// TIA Portal V16 export
// export: Created 2023-03-29T11:03:29.1138509Z, ExportSetting WithDefaults, DisplayName Totally Integrated Automation Portal, DisplayVersion V16 Update 6, DisplayName TIA Portal Version Control Interface, DisplayVersion V16 Update 2, DisplayName TIA Portal Openness, DisplayVersion V16 Update 6, DisplayName STEP 7 Professional, DisplayVersion V16 Update 6, DisplayName STEP 7 Safety, DisplayVersion V16, DisplayName WinCC Advanced, DisplayVersion V16 Update 6
FUNCTION "Sterowniki napędów" : Void   // FC7, LAD
TITLE = Sterowniki
{ S7_Optimized_Access := 'TRUE' }
AUTHOR : rtecmer
VERSION : 0.1
// Sterownik napędów zasuw Z1-Z9
// stored: AutoNumber true, IsIECCheckEnabled false, SetENOAutomatically false, UDAEnableTagReadback false
BEGIN

REGION Network 2: Sterowanie Zasuwą Z10 - Położenie
   // Funkcja zawiera kontrolę czasu jazdy na pozycję ustawiony czas 120sek
   // po upływie czasu nastapi alarm i przełączenie w trym manual
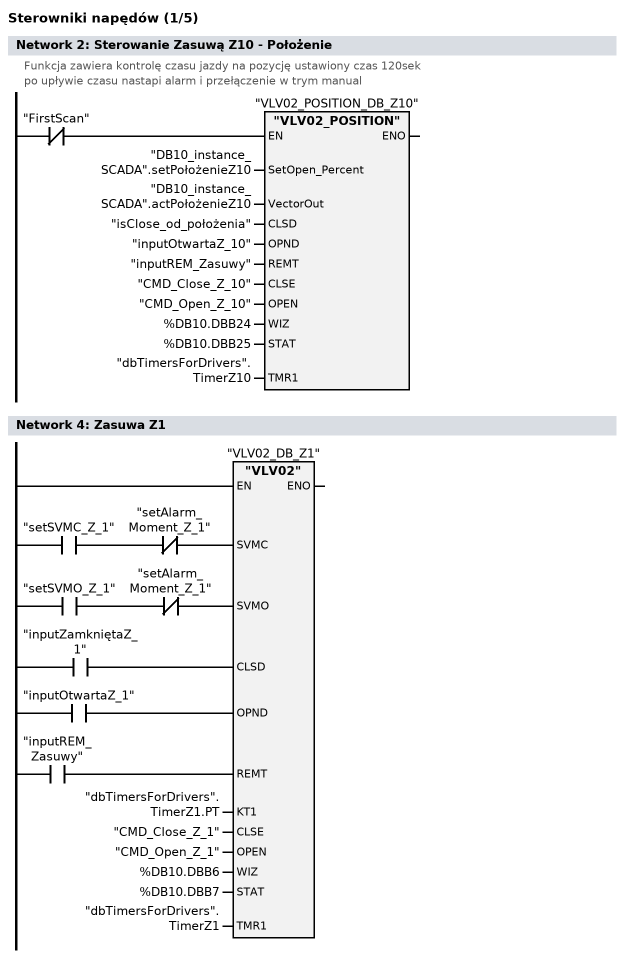
   RUNG wire#powerrail
      I_Contact( "FirstScan" )
      "VLV02_POSITION_DB_Z10"(SetOpen_Percent := "DB10_instance_SCADA".setPołożenieZ10, VectorOut := "DB10_instance_SCADA".actPołożenieZ10, CLSD := "isClose_od_położenia", OPND := "inputOtwartaZ_10", REMT := "inputREM_Zasuwy", CLSE := "CMD_Close_Z_10", OPEN := "CMD_Open_Z_10", WIZ := %DB10.DBB24, STAT := %DB10.DBB25, TMR1 := "dbTimersForDrivers".TimerZ10)
   END_RUNG
   // the same network as SCL:
   IF NOT "FirstScan" THEN
       "VLV02_POSITION_DB_Z10"(SetOpen_Percent := "DB10_instance_SCADA".setPołożenieZ10,   // "VLV02_POSITION"
                               VectorOut := "DB10_instance_SCADA".actPołożenieZ10,
                               CLSD := "isClose_od_położenia",
                               OPND := "inputOtwartaZ_10",
                               REMT := "inputREM_Zasuwy",
                               CLSE := "CMD_Close_Z_10",
                               OPEN := "CMD_Open_Z_10",
                               WIZ := %DB10.DBB24,
                               STAT := %DB10.DBB25,
                               TMR1 := "dbTimersForDrivers".TimerZ10);
   END_IF;
END_REGION

REGION Network 4: Zasuwa Z1
   RUNG wire#powerrail
      "VLV02_DB_Z1"(SVMC := wire#w1, SVMO := wire#w2, CLSD := wire#w3, OPND := wire#w4, REMT := wire#w5, KT1 := "dbTimersForDrivers".TimerZ1.PT, CLSE := "CMD_Close_Z_1", OPEN := "CMD_Open_Z_1", WIZ := %DB10.DBB6, STAT := %DB10.DBB7, TMR1 := "dbTimersForDrivers".TimerZ1)
   END_RUNG
   RUNG wire#powerrail
      Contact( "setSVMC_Z_1" )
      I_Contact( "setAlarm_Moment_Z_1" )
   END_RUNG wire#w1
   RUNG wire#powerrail
      Contact( "setSVMO_Z_1" )
      I_Contact( "setAlarm_Moment_Z_1" )
   END_RUNG wire#w2
   RUNG wire#powerrail
      Contact( "inputZamkniętaZ_1" )
   END_RUNG wire#w3
   RUNG wire#powerrail
      Contact( "inputOtwartaZ_1" )
   END_RUNG wire#w4
   RUNG wire#powerrail
      Contact( "inputREM_Zasuwy" )
   END_RUNG wire#w5
   // the same network as SCL:
   "VLV02_DB_Z1"(SVMC := "setSVMC_Z_1" AND NOT "setAlarm_Moment_Z_1",   // "VLV02"
                 SVMO := "setSVMO_Z_1" AND NOT "setAlarm_Moment_Z_1",
                 CLSD := "inputZamkniętaZ_1",
                 OPND := "inputOtwartaZ_1",
                 REMT := "inputREM_Zasuwy",
                 KT1 := "dbTimersForDrivers".TimerZ1.PT,
                 CLSE := "CMD_Close_Z_1",
                 OPEN := "CMD_Open_Z_1",
                 WIZ := %DB10.DBB6,
                 STAT := %DB10.DBB7,
                 TMR1 := "dbTimersForDrivers".TimerZ1);
END_REGION

REGION Network 5: Zasuwa Z2
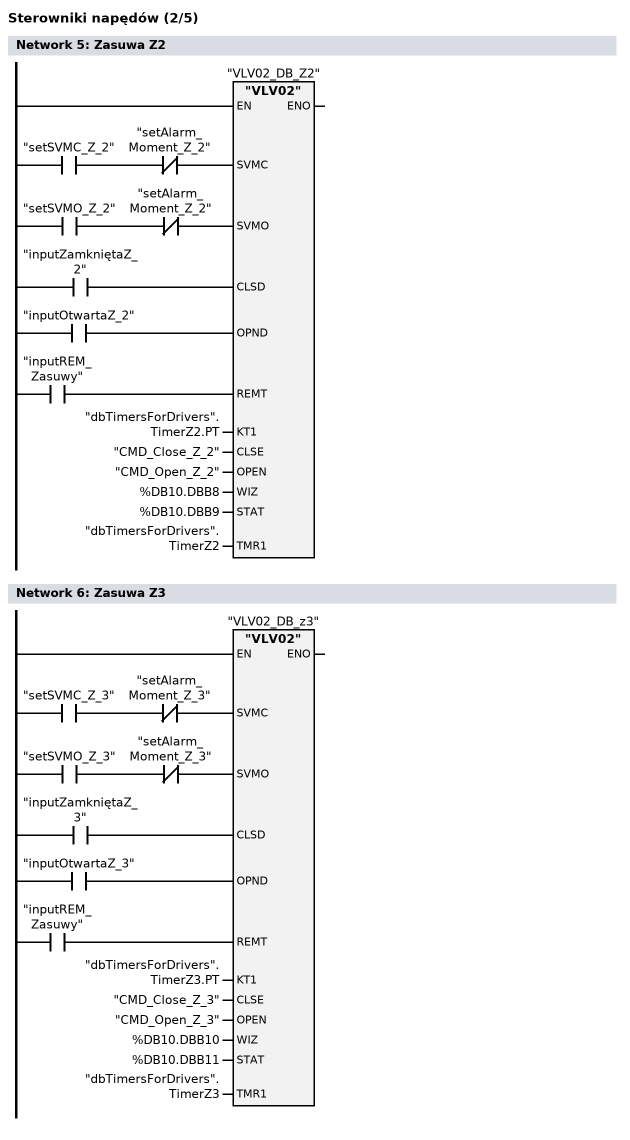
   RUNG wire#powerrail
      "VLV02_DB_Z2"(SVMC := wire#w1, SVMO := wire#w2, CLSD := wire#w3, OPND := wire#w4, REMT := wire#w5, KT1 := "dbTimersForDrivers".TimerZ2.PT, CLSE := "CMD_Close_Z_2", OPEN := "CMD_Open_Z_2", WIZ := %DB10.DBB8, STAT := %DB10.DBB9, TMR1 := "dbTimersForDrivers".TimerZ2)
   END_RUNG
   RUNG wire#powerrail
      Contact( "setSVMC_Z_2" )
      I_Contact( "setAlarm_Moment_Z_2" )
   END_RUNG wire#w1
   RUNG wire#powerrail
      Contact( "setSVMO_Z_2" )
      I_Contact( "setAlarm_Moment_Z_2" )
   END_RUNG wire#w2
   RUNG wire#powerrail
      Contact( "inputZamkniętaZ_2" )
   END_RUNG wire#w3
   RUNG wire#powerrail
      Contact( "inputOtwartaZ_2" )
   END_RUNG wire#w4
   RUNG wire#powerrail
      Contact( "inputREM_Zasuwy" )
   END_RUNG wire#w5
   // the same network as SCL:
   "VLV02_DB_Z2"(SVMC := "setSVMC_Z_2" AND NOT "setAlarm_Moment_Z_2",   // "VLV02"
                 SVMO := "setSVMO_Z_2" AND NOT "setAlarm_Moment_Z_2",
                 CLSD := "inputZamkniętaZ_2",
                 OPND := "inputOtwartaZ_2",
                 REMT := "inputREM_Zasuwy",
                 KT1 := "dbTimersForDrivers".TimerZ2.PT,
                 CLSE := "CMD_Close_Z_2",
                 OPEN := "CMD_Open_Z_2",
                 WIZ := %DB10.DBB8,
                 STAT := %DB10.DBB9,
                 TMR1 := "dbTimersForDrivers".TimerZ2);
END_REGION

REGION Network 6: Zasuwa Z3
   RUNG wire#powerrail
      "VLV02_DB_z3"(SVMC := wire#w1, SVMO := wire#w2, CLSD := wire#w3, OPND := wire#w4, REMT := wire#w5, KT1 := "dbTimersForDrivers".TimerZ3.PT, CLSE := "CMD_Close_Z_3", OPEN := "CMD_Open_Z_3", WIZ := %DB10.DBB10, STAT := %DB10.DBB11, TMR1 := "dbTimersForDrivers".TimerZ3)
   END_RUNG
   RUNG wire#powerrail
      Contact( "setSVMC_Z_3" )
      I_Contact( "setAlarm_Moment_Z_3" )
   END_RUNG wire#w1
   RUNG wire#powerrail
      Contact( "setSVMO_Z_3" )
      I_Contact( "setAlarm_Moment_Z_3" )
   END_RUNG wire#w2
   RUNG wire#powerrail
      Contact( "inputZamkniętaZ_3" )
   END_RUNG wire#w3
   RUNG wire#powerrail
      Contact( "inputOtwartaZ_3" )
   END_RUNG wire#w4
   RUNG wire#powerrail
      Contact( "inputREM_Zasuwy" )
   END_RUNG wire#w5
   // the same network as SCL:
   "VLV02_DB_z3"(SVMC := "setSVMC_Z_3" AND NOT "setAlarm_Moment_Z_3",   // "VLV02"
                 SVMO := "setSVMO_Z_3" AND NOT "setAlarm_Moment_Z_3",
                 CLSD := "inputZamkniętaZ_3",
                 OPND := "inputOtwartaZ_3",
                 REMT := "inputREM_Zasuwy",
                 KT1 := "dbTimersForDrivers".TimerZ3.PT,
                 CLSE := "CMD_Close_Z_3",
                 OPEN := "CMD_Open_Z_3",
                 WIZ := %DB10.DBB10,
                 STAT := %DB10.DBB11,
                 TMR1 := "dbTimersForDrivers".TimerZ3);
END_REGION

REGION Network 7: Zasuwa Z4
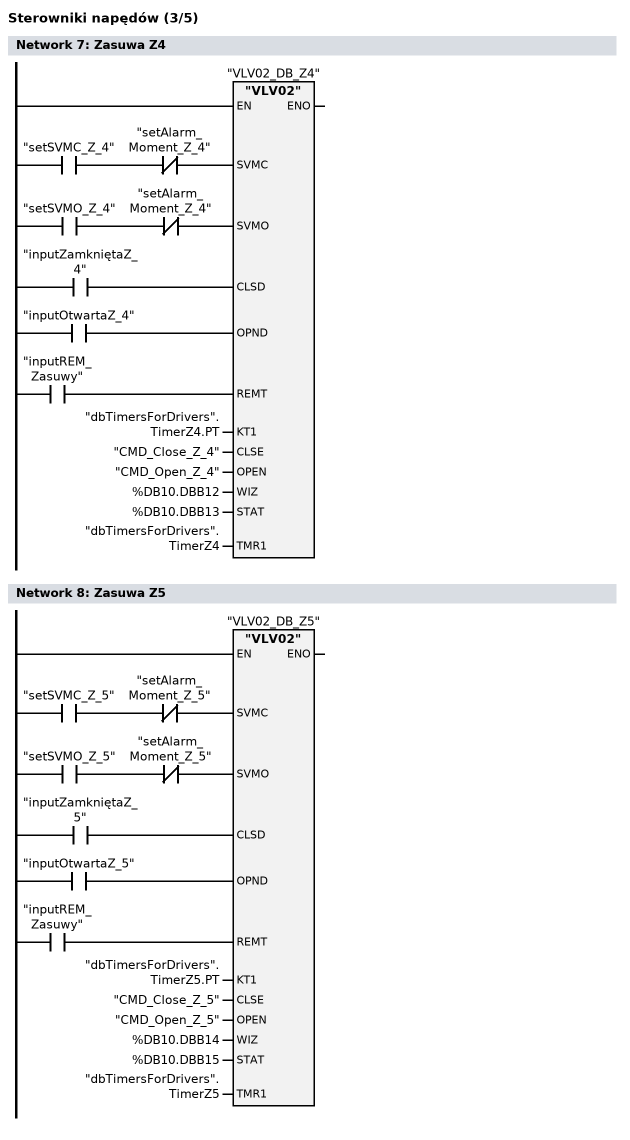
   RUNG wire#powerrail
      "VLV02_DB_Z4"(SVMC := wire#w1, SVMO := wire#w2, CLSD := wire#w3, OPND := wire#w4, REMT := wire#w5, KT1 := "dbTimersForDrivers".TimerZ4.PT, CLSE := "CMD_Close_Z_4", OPEN := "CMD_Open_Z_4", WIZ := %DB10.DBB12, STAT := %DB10.DBB13, TMR1 := "dbTimersForDrivers".TimerZ4)
   END_RUNG
   RUNG wire#powerrail
      Contact( "setSVMC_Z_4" )
      I_Contact( "setAlarm_Moment_Z_4" )
   END_RUNG wire#w1
   RUNG wire#powerrail
      Contact( "setSVMO_Z_4" )
      I_Contact( "setAlarm_Moment_Z_4" )
   END_RUNG wire#w2
   RUNG wire#powerrail
      Contact( "inputZamkniętaZ_4" )
   END_RUNG wire#w3
   RUNG wire#powerrail
      Contact( "inputOtwartaZ_4" )
   END_RUNG wire#w4
   RUNG wire#powerrail
      Contact( "inputREM_Zasuwy" )
   END_RUNG wire#w5
   // the same network as SCL:
   "VLV02_DB_Z4"(SVMC := "setSVMC_Z_4" AND NOT "setAlarm_Moment_Z_4",   // "VLV02"
                 SVMO := "setSVMO_Z_4" AND NOT "setAlarm_Moment_Z_4",
                 CLSD := "inputZamkniętaZ_4",
                 OPND := "inputOtwartaZ_4",
                 REMT := "inputREM_Zasuwy",
                 KT1 := "dbTimersForDrivers".TimerZ4.PT,
                 CLSE := "CMD_Close_Z_4",
                 OPEN := "CMD_Open_Z_4",
                 WIZ := %DB10.DBB12,
                 STAT := %DB10.DBB13,
                 TMR1 := "dbTimersForDrivers".TimerZ4);
END_REGION

REGION Network 8: Zasuwa Z5
   RUNG wire#powerrail
      "VLV02_DB_Z5"(SVMC := wire#w1, SVMO := wire#w2, CLSD := wire#w3, OPND := wire#w4, REMT := wire#w5, KT1 := "dbTimersForDrivers".TimerZ5.PT, CLSE := "CMD_Close_Z_5", OPEN := "CMD_Open_Z_5", WIZ := %DB10.DBB14, STAT := %DB10.DBB15, TMR1 := "dbTimersForDrivers".TimerZ5)
   END_RUNG
   RUNG wire#powerrail
      Contact( "setSVMC_Z_5" )
      I_Contact( "setAlarm_Moment_Z_5" )
   END_RUNG wire#w1
   RUNG wire#powerrail
      Contact( "setSVMO_Z_5" )
      I_Contact( "setAlarm_Moment_Z_5" )
   END_RUNG wire#w2
   RUNG wire#powerrail
      Contact( "inputZamkniętaZ_5" )
   END_RUNG wire#w3
   RUNG wire#powerrail
      Contact( "inputOtwartaZ_5" )
   END_RUNG wire#w4
   RUNG wire#powerrail
      Contact( "inputREM_Zasuwy" )
   END_RUNG wire#w5
   // the same network as SCL:
   "VLV02_DB_Z5"(SVMC := "setSVMC_Z_5" AND NOT "setAlarm_Moment_Z_5",   // "VLV02"
                 SVMO := "setSVMO_Z_5" AND NOT "setAlarm_Moment_Z_5",
                 CLSD := "inputZamkniętaZ_5",
                 OPND := "inputOtwartaZ_5",
                 REMT := "inputREM_Zasuwy",
                 KT1 := "dbTimersForDrivers".TimerZ5.PT,
                 CLSE := "CMD_Close_Z_5",
                 OPEN := "CMD_Open_Z_5",
                 WIZ := %DB10.DBB14,
                 STAT := %DB10.DBB15,
                 TMR1 := "dbTimersForDrivers".TimerZ5);
END_REGION

REGION Network 9: Zasuwa Z6
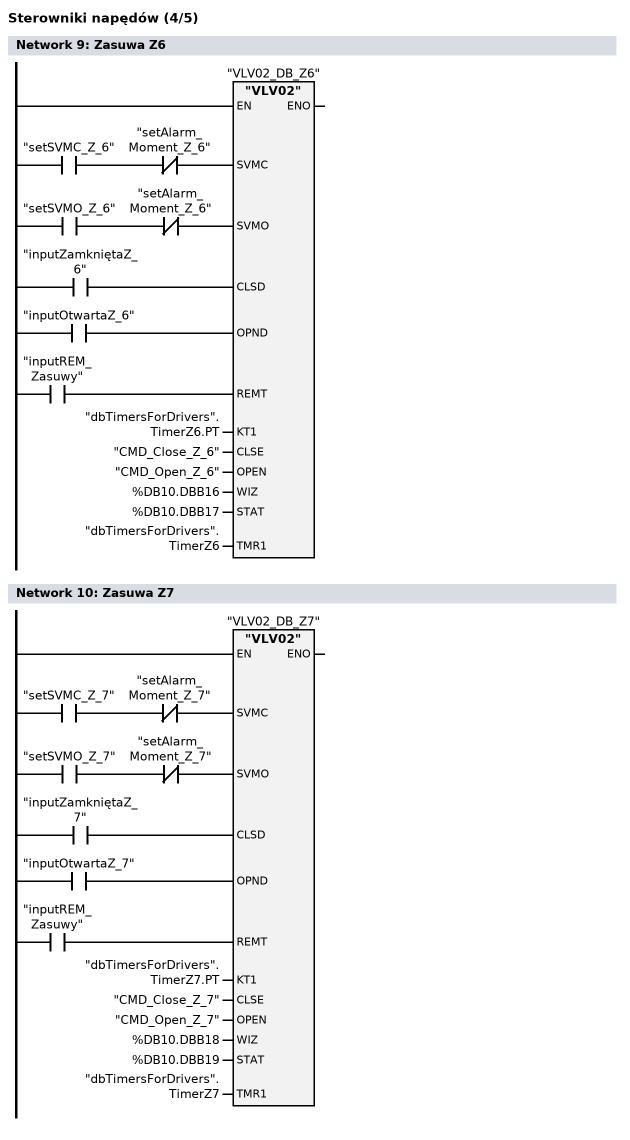
   RUNG wire#powerrail
      "VLV02_DB_Z6"(SVMC := wire#w1, SVMO := wire#w2, CLSD := wire#w3, OPND := wire#w4, REMT := wire#w5, KT1 := "dbTimersForDrivers".TimerZ6.PT, CLSE := "CMD_Close_Z_6", OPEN := "CMD_Open_Z_6", WIZ := %DB10.DBB16, STAT := %DB10.DBB17, TMR1 := "dbTimersForDrivers".TimerZ6)
   END_RUNG
   RUNG wire#powerrail
      Contact( "setSVMC_Z_6" )
      I_Contact( "setAlarm_Moment_Z_6" )
   END_RUNG wire#w1
   RUNG wire#powerrail
      Contact( "setSVMO_Z_6" )
      I_Contact( "setAlarm_Moment_Z_6" )
   END_RUNG wire#w2
   RUNG wire#powerrail
      Contact( "inputZamkniętaZ_6" )
   END_RUNG wire#w3
   RUNG wire#powerrail
      Contact( "inputOtwartaZ_6" )
   END_RUNG wire#w4
   RUNG wire#powerrail
      Contact( "inputREM_Zasuwy" )
   END_RUNG wire#w5
   // the same network as SCL:
   "VLV02_DB_Z6"(SVMC := "setSVMC_Z_6" AND NOT "setAlarm_Moment_Z_6",   // "VLV02"
                 SVMO := "setSVMO_Z_6" AND NOT "setAlarm_Moment_Z_6",
                 CLSD := "inputZamkniętaZ_6",
                 OPND := "inputOtwartaZ_6",
                 REMT := "inputREM_Zasuwy",
                 KT1 := "dbTimersForDrivers".TimerZ6.PT,
                 CLSE := "CMD_Close_Z_6",
                 OPEN := "CMD_Open_Z_6",
                 WIZ := %DB10.DBB16,
                 STAT := %DB10.DBB17,
                 TMR1 := "dbTimersForDrivers".TimerZ6);
END_REGION

REGION Network 10: Zasuwa Z7
   RUNG wire#powerrail
      "VLV02_DB_Z7"(SVMC := wire#w1, SVMO := wire#w2, CLSD := wire#w3, OPND := wire#w4, REMT := wire#w5, KT1 := "dbTimersForDrivers".TimerZ7.PT, CLSE := "CMD_Close_Z_7", OPEN := "CMD_Open_Z_7", WIZ := %DB10.DBB18, STAT := %DB10.DBB19, TMR1 := "dbTimersForDrivers".TimerZ7)
   END_RUNG
   RUNG wire#powerrail
      Contact( "setSVMC_Z_7" )
      I_Contact( "setAlarm_Moment_Z_7" )
   END_RUNG wire#w1
   RUNG wire#powerrail
      Contact( "setSVMO_Z_7" )
      I_Contact( "setAlarm_Moment_Z_7" )
   END_RUNG wire#w2
   RUNG wire#powerrail
      Contact( "inputZamkniętaZ_7" )
   END_RUNG wire#w3
   RUNG wire#powerrail
      Contact( "inputOtwartaZ_7" )
   END_RUNG wire#w4
   RUNG wire#powerrail
      Contact( "inputREM_Zasuwy" )
   END_RUNG wire#w5
   // the same network as SCL:
   "VLV02_DB_Z7"(SVMC := "setSVMC_Z_7" AND NOT "setAlarm_Moment_Z_7",   // "VLV02"
                 SVMO := "setSVMO_Z_7" AND NOT "setAlarm_Moment_Z_7",
                 CLSD := "inputZamkniętaZ_7",
                 OPND := "inputOtwartaZ_7",
                 REMT := "inputREM_Zasuwy",
                 KT1 := "dbTimersForDrivers".TimerZ7.PT,
                 CLSE := "CMD_Close_Z_7",
                 OPEN := "CMD_Open_Z_7",
                 WIZ := %DB10.DBB18,
                 STAT := %DB10.DBB19,
                 TMR1 := "dbTimersForDrivers".TimerZ7);
END_REGION

REGION Network 11: Zasuwa Z8
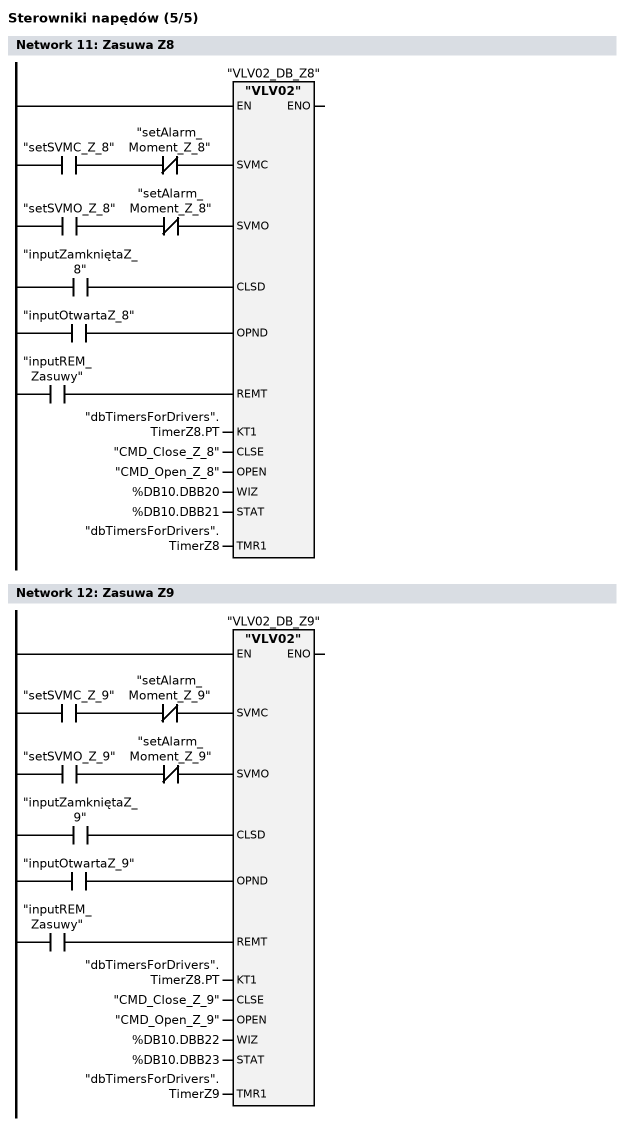
   RUNG wire#powerrail
      "VLV02_DB_Z8"(SVMC := wire#w1, SVMO := wire#w2, CLSD := wire#w3, OPND := wire#w4, REMT := wire#w5, KT1 := "dbTimersForDrivers".TimerZ8.PT, CLSE := "CMD_Close_Z_8", OPEN := "CMD_Open_Z_8", WIZ := %DB10.DBB20, STAT := %DB10.DBB21, TMR1 := "dbTimersForDrivers".TimerZ8)
   END_RUNG
   RUNG wire#powerrail
      Contact( "setSVMC_Z_8" )
      I_Contact( "setAlarm_Moment_Z_8" )
   END_RUNG wire#w1
   RUNG wire#powerrail
      Contact( "setSVMO_Z_8" )
      I_Contact( "setAlarm_Moment_Z_8" )
   END_RUNG wire#w2
   RUNG wire#powerrail
      Contact( "inputZamkniętaZ_8" )
   END_RUNG wire#w3
   RUNG wire#powerrail
      Contact( "inputOtwartaZ_8" )
   END_RUNG wire#w4
   RUNG wire#powerrail
      Contact( "inputREM_Zasuwy" )
   END_RUNG wire#w5
   // the same network as SCL:
   "VLV02_DB_Z8"(SVMC := "setSVMC_Z_8" AND NOT "setAlarm_Moment_Z_8",   // "VLV02"
                 SVMO := "setSVMO_Z_8" AND NOT "setAlarm_Moment_Z_8",
                 CLSD := "inputZamkniętaZ_8",
                 OPND := "inputOtwartaZ_8",
                 REMT := "inputREM_Zasuwy",
                 KT1 := "dbTimersForDrivers".TimerZ8.PT,
                 CLSE := "CMD_Close_Z_8",
                 OPEN := "CMD_Open_Z_8",
                 WIZ := %DB10.DBB20,
                 STAT := %DB10.DBB21,
                 TMR1 := "dbTimersForDrivers".TimerZ8);
END_REGION

REGION Network 12: Zasuwa Z9
   RUNG wire#powerrail
      "VLV02_DB_Z9"(SVMC := wire#w1, SVMO := wire#w2, CLSD := wire#w3, OPND := wire#w4, REMT := wire#w5, KT1 := "dbTimersForDrivers".TimerZ8.PT, CLSE := "CMD_Close_Z_9", OPEN := "CMD_Open_Z_9", WIZ := %DB10.DBB22, STAT := %DB10.DBB23, TMR1 := "dbTimersForDrivers".TimerZ9)
   END_RUNG
   RUNG wire#powerrail
      Contact( "setSVMC_Z_9" )
      I_Contact( "setAlarm_Moment_Z_9" )
   END_RUNG wire#w1
   RUNG wire#powerrail
      Contact( "setSVMO_Z_9" )
      I_Contact( "setAlarm_Moment_Z_9" )
   END_RUNG wire#w2
   RUNG wire#powerrail
      Contact( "inputZamkniętaZ_9" )
   END_RUNG wire#w3
   RUNG wire#powerrail
      Contact( "inputOtwartaZ_9" )
   END_RUNG wire#w4
   RUNG wire#powerrail
      Contact( "inputREM_Zasuwy" )
   END_RUNG wire#w5
   // the same network as SCL:
   "VLV02_DB_Z9"(SVMC := "setSVMC_Z_9" AND NOT "setAlarm_Moment_Z_9",   // "VLV02"
                 SVMO := "setSVMO_Z_9" AND NOT "setAlarm_Moment_Z_9",
                 CLSD := "inputZamkniętaZ_9",
                 OPND := "inputOtwartaZ_9",
                 REMT := "inputREM_Zasuwy",
                 KT1 := "dbTimersForDrivers".TimerZ8.PT,
                 CLSE := "CMD_Close_Z_9",
                 OPEN := "CMD_Open_Z_9",
                 WIZ := %DB10.DBB22,
                 STAT := %DB10.DBB23,
                 TMR1 := "dbTimersForDrivers".TimerZ9);
END_REGION
END_FUNCTION
